	DATA_BLOCK DB381
	TITLE =DBG281M  ELEVATOR 9002 AFTER KILN
	//COPYRIGHT:    (C) 2009  BUHLER AG, CH-9240 UZWIL, SWITZERLAND
	//
	//PRODUCT:      WinCoS_BIW01_09
	//
	//TITLE:        ELEVATOR 9002 AFTER KILN
	//                Machine group DB
	//                Maschinengruppen-DB
	//
	//-------------------------------------------------------------------------
	//
	//IDENT:        AUTHOR:             DEPT:             DATE:
	//
	//P01_DB381.1.0 K.Renz              CSB41             13.Jan.2010
	//              1st Release
	//
	//-------------------------------------------------------------------------
	//
	//PURPOSE:
	//
	//MANUAL :
	//
	//RESTRICTIONS:
	//
	//-------------------------------------------------------------------------
	AUTHOR  : KR
	FAMILY  : USW
	NAME    : DBG281M
	VERSION : 00.00

	FB381
	BEGIN
	      #Gr.Par.ParObjectNo 	:=28100;
	      #Gr.Par.ParIdling      	:=2;
	      #Gr.Par.ParMgr	        :=True;
	      #Gr.Par.ParWgr	        :=False;
	      #Gr.Par.ParGgr	        :=False;
	      #Gr.Par.ParEmptyingTime 	:=0;
	      #Gr.Par.ParHornCode       :=12;
	//Parameter =A-3930-MXZ01MA : ELEVATOR
	      #A_3930_MXZ01MA.Ma.Par.ParObjectNo                                     :=28101;
	      #A_3930_MXZ01MA.Ma.Par.ParWithMon3                                     :=True;
	      #A_3930_MXZ01MA.Ma.Par.ParWithMon4                                     :=True;
	      #A_3930_MXZ01MA.Ma.Par.ParMon1IsHL                                     :=True;
	      #A_3930_MXZ01MA.Ma.Par.ParMon1IsLS                                     :=False;
	      #A_3930_MXZ01MA.Ma.Par.ParMon1StopByFault                              :=True;
	      #A_3930_MXZ01MA.Ma.Par.ParMon2IsLS                                     :=True;
	      #A_3930_MXZ01MA.Ma.Par.ParMon3IsLS                                     :=True;
	      #A_3930_MXZ01MA.Ma.Par.ParMon4AsWarning                                :=False;
	      #A_3930_MXZ01MA.Ma.Par.ParMon4StopByFault                              :=True;
	      #A_3930_MXZ01MA.Ma.Par.ParMon4IsLS                                     :=False;
	      #A_3930_MXZ01MA.Ma.Par.ParWithMon1                                     :=True;
	      #A_3930_MXZ01MA.Ma.Par.ParWithMon5                                     :=False;
	      #A_3930_MXZ01MA.Ma.Par.ParWithMon6                                     :=False;
	      #A_3930_MXZ01MA.Ma.Par.ParEBM                                          :=False;
	      #A_3930_MXZ01MA.Ma.Par.ParMon4IsSM                                     :=True;
	//
	//Parameter A_3930_MXZ01MA.=A-3930-BLH31 : STOWING DETECTOR DISCHARGE
	      #A_3930_MXZ01MA.A_3930_BLH31.Par.ParObjectNo                             :=28102;
	      #A_3930_MXZ01MA.A_3930_BLH31.Par.ParMsgType                              :=7165;
	      #A_3930_MXZ01MA.A_3930_BLH31.Par.ParHornCode                             :=12;
	      #A_3930_MXZ01MA.A_3930_BLH31.Par.ParDelayChange                          :=20;
	      #A_3930_MXZ01MA.A_3930_BLH31.Par.ParDelayCovered                         :=10;
	      #A_3930_MXZ01MA.A_3930_BLH31.Par.ParDelayUncovered                       :=30;
	      #A_3930_MXZ01MA.A_3930_BLH31.Par.ParTimeoutCovered                       :=0;
	      #A_3930_MXZ01MA.A_3930_BLH31.Par.ParTimeoutUncovered                     :=0;
	      #A_3930_MXZ01MA.A_3930_BLH31.Par.ParLogOff                               :=False;
	      #A_3930_MXZ01MA.A_3930_BLH31.Par.Par2WorkingCond                         :=False;
	      #A_3930_MXZ01MA.A_3930_BLH31.Par.ParFaultRetry                           :=False;
	      #A_3930_MXZ01MA.A_3930_BLH31.Par.ParBinLevel                             :=False;
	//
	//Parameter A_3930_MXZ01MA.=A-3930-SHE29 : EMERGENCY-OFF ELEVATOR
	      #A_3930_MXZ01MA.A_3930_SHE29.Par.ParObjectNo                             :=28103;
	      #A_3930_MXZ01MA.A_3930_SHE29.Par.ParMsgType                              :=7136;
	      #A_3930_MXZ01MA.A_3930_SHE29.Par.ParHornCode                             :=12;
	      #A_3930_MXZ01MA.A_3930_SHE29.Par.ParDelayChange                          :=20;
	      #A_3930_MXZ01MA.A_3930_SHE29.Par.ParDelayTrue                            :=10;
	      #A_3930_MXZ01MA.A_3930_SHE29.Par.ParDelayFalse                           :=0;
	      #A_3930_MXZ01MA.A_3930_SHE29.Par.ParTimeoutTrue                          :=0;
	      #A_3930_MXZ01MA.A_3930_SHE29.Par.ParTimeoutFalse                         :=0;
	      #A_3930_MXZ01MA.A_3930_SHE29.Par.ParLogOff                               :=False;
	      #A_3930_MXZ01MA.A_3930_SHE29.Par.Par2WorkingCond                         :=False;
	      #A_3930_MXZ01MA.A_3930_SHE29.Par.ParFaultRetry                           :=False;
	      #A_3930_MXZ01MA.A_3930_SHE29.Par.ParBinLevel                             :=False;
	//
	//Parameter A_3930_MXZ01MA.=A-3930-SHE28 : EMERGENCY-OFF ELEVATOR
	      #A_3930_MXZ01MA.A_3930_SHE28.Par.ParObjectNo                             :=28104;
	      #A_3930_MXZ01MA.A_3930_SHE28.Par.ParMsgType                              :=7136;
	      #A_3930_MXZ01MA.A_3930_SHE28.Par.ParHornCode                             :=12;
	      #A_3930_MXZ01MA.A_3930_SHE28.Par.ParDelayChange                          :=20;
	      #A_3930_MXZ01MA.A_3930_SHE28.Par.ParDelayTrue                            :=10;
	      #A_3930_MXZ01MA.A_3930_SHE28.Par.ParDelayFalse                           :=0;
	      #A_3930_MXZ01MA.A_3930_SHE28.Par.ParTimeoutTrue                          :=0;
	      #A_3930_MXZ01MA.A_3930_SHE28.Par.ParTimeoutFalse                         :=0;
	      #A_3930_MXZ01MA.A_3930_SHE28.Par.ParLogOff                               :=False;
	      #A_3930_MXZ01MA.A_3930_SHE28.Par.Par2WorkingCond                         :=False;
	      #A_3930_MXZ01MA.A_3930_SHE28.Par.ParFaultRetry                           :=False;
	      #A_3930_MXZ01MA.A_3930_SHE28.Par.ParBinLevel                             :=False;
	//
	//Parameter A_3930_MXZ01MA.=A-3930-BSA07 : SPEED CONTROL
	      #A_3930_MXZ01MA.A_3930_BSA07.Par.ParObjectNo                             :=28105;
	      #A_3930_MXZ01MA.A_3930_BSA07.Par.ParMsgType                              :=7135;
	      #A_3930_MXZ01MA.A_3930_BSA07.Par.ParHornCode                             :=12;
	      #A_3930_MXZ01MA.A_3930_BSA07.Par.ParDelayChange                          :=0;
	      #A_3930_MXZ01MA.A_3930_BSA07.Par.ParDelayTrue                            :=10;
	      #A_3930_MXZ01MA.A_3930_BSA07.Par.ParDelayFalse                           :=0;
	      #A_3930_MXZ01MA.A_3930_BSA07.Par.ParTimeoutTrue                          :=50;
	      #A_3930_MXZ01MA.A_3930_BSA07.Par.ParTimeoutFalse                         :=0;
	      #A_3930_MXZ01MA.A_3930_BSA07.Par.ParLogOff                               :=False;
	      #A_3930_MXZ01MA.A_3930_BSA07.Par.Par2WorkingCond                         :=True;
	      #A_3930_MXZ01MA.A_3930_BSA07.Par.ParFaultRetry                           :=False;
	      #A_3930_MXZ01MA.A_3930_BSA07.Par.ParBinLevel                             :=False;
	//
	//Parameter A_3930_MXZ01MA.=A-3930-MXZ01 : ELEVATOR
	      #A_3930_MXZ01MA.A_3930_MXZ01.Par.ParObjectNo                             :=28106;
	      #A_3930_MXZ01MA.A_3930_MXZ01.Par.ParMsgType                              :=7053;
	      #A_3930_MXZ01MA.A_3930_MXZ01.Par.ParHornCode                             :=12;
	      #A_3930_MXZ01MA.A_3930_MXZ01.Par.ParMonTime                              :=20;
	      #A_3930_MXZ01MA.A_3930_MXZ01.Par.ParStartingTime                         :=20;
	      #A_3930_MXZ01MA.A_3930_MXZ01.Par.ParStoppingTime                         :=0;
	      #A_3930_MXZ01MA.A_3930_MXZ01.Par.ParIdlingTime                           :=0;
	      #A_3930_MXZ01MA.A_3930_MXZ01.Par.ParDelayTime                            :=10;
	      #A_3930_MXZ01MA.A_3930_MXZ01.Par.ParLogOff                               :=False;
	      #A_3930_MXZ01MA.A_3930_MXZ01.Par.ParManual                               :=True;
	      #A_3930_MXZ01MA.A_3930_MXZ01.Par.ParRestartDelay                         :=False;
	      #A_3930_MXZ01MA.A_3930_MXZ01.Par.Par2Speed                               :=False;
	      #A_3930_MXZ01MA.A_3930_MXZ01.Par.ParHeavyStartup                         :=False;
	//
	//
	//Parameter =A-3932-MXZ01MA : FILTER ASPIRATION ELEVATOR
	      #A_3932_MXZ01MA.Ma.Par.ParObjectNo                                     :=28107;
	      #A_3932_MXZ01MA.Ma.Par.ParWithAirlock                                  :=False;
	      #A_3932_MXZ01MA.Ma.Par.ParWithFan                                      :=True;
	      #A_3932_MXZ01MA.Ma.Par.ParWithFilter                                   :=True;
	      #A_3932_MXZ01MA.Ma.Par.ParWithARF                                      :=False;
	      #A_3932_MXZ01MA.Ma.Par.ParWithLSDoor                                   :=False;
	      #A_3932_MXZ01MA.Ma.Par.ParWithPressure                                 :=False;
	      #A_3932_MXZ01MA.Ma.Par.ParWithHLAirlock                                :=False;
	      #A_3932_MXZ01MA.Ma.Par.ParWithDischarger                               :=False;
	      #A_3932_MXZ01MA.Ma.Par.ParVibroOnTime                                  :=0;
	      #A_3932_MXZ01MA.Ma.Par.ParVibroOffTime                                 :=0;
	//
	//Parameter A_3932_MXZ01MA.=A-3932-MXZ01 : FAN DRIVE
	      #A_3932_MXZ01MA.A_3932_MXZ01.Par.ParObjectNo                             :=28108;
	      #A_3932_MXZ01MA.A_3932_MXZ01.Par.ParMsgType                              :=7053;
	      #A_3932_MXZ01MA.A_3932_MXZ01.Par.ParHornCode                             :=12;
	      #A_3932_MXZ01MA.A_3932_MXZ01.Par.ParMonTime                              :=20;
	      #A_3932_MXZ01MA.A_3932_MXZ01.Par.ParStartingTime                         :=20;
	      #A_3932_MXZ01MA.A_3932_MXZ01.Par.ParStoppingTime                         :=0;
	      #A_3932_MXZ01MA.A_3932_MXZ01.Par.ParIdlingTime                           :=0;
	      #A_3932_MXZ01MA.A_3932_MXZ01.Par.ParDelayTime                            :=10;
	      #A_3932_MXZ01MA.A_3932_MXZ01.Par.ParLogOff                               :=False;
	      #A_3932_MXZ01MA.A_3932_MXZ01.Par.ParManual                               :=True;
	      #A_3932_MXZ01MA.A_3932_MXZ01.Par.ParRestartDelay                         :=False;
	      #A_3932_MXZ01MA.A_3932_MXZ01.Par.Par2Speed                               :=False;
	      #A_3932_MXZ01MA.A_3932_MXZ01.Par.ParHeavyStartup                         :=False;
	//
	//Parameter A_3932_MXZ01MA.=A-3931-KFC10 : FILTER ASPIRATION
	      #A_3932_MXZ01MA.A_3931_KFC10.Par.ParObjectNo                             :=28109;
	      #A_3932_MXZ01MA.A_3931_KFC10.Par.ParMsgType                              :=7002;
	      #A_3932_MXZ01MA.A_3931_KFC10.Par.ParHornCode                             :=12;
	      #A_3932_MXZ01MA.A_3931_KFC10.Par.ParOnTime                               :=50;
	      #A_3932_MXZ01MA.A_3931_KFC10.Par.ParOffTime                              :=0;
	      #A_3932_MXZ01MA.A_3931_KFC10.Par.ParIdlingTime                           :=3000;
	      #A_3932_MXZ01MA.A_3931_KFC10.Par.ParDelayTime                            :=0;
	      #A_3932_MXZ01MA.A_3931_KFC10.Par.ParLogOff                               :=False;
	      #A_3932_MXZ01MA.A_3931_KFC10.Par.ParManual                               :=True;
	      #A_3932_MXZ01MA.A_3931_KFC10.Par.ParContinuous                           :=True;
	      #A_3932_MXZ01MA.A_3931_KFC10.Par.ParPulse                                :=False;
	      #A_3932_MXZ01MA.A_3931_KFC10.Par.ParPulsing                              :=False;
	      #A_3932_MXZ01MA.A_3931_KFC10.Par.ParFilter                               :=True;
	//
	//
	//Parameter =A-3930-KCL01 : RESET DISTURBANCE ELEVATOR
	      #A_3930_KCL01.Par.ParObjectNo                             :=28110;
	      #A_3930_KCL01.Par.ParMsgType                              :=7154;
	      #A_3930_KCL01.Par.ParHornCode                             :=12;
	      #A_3930_KCL01.Par.ParDelayChange                          :=20;
	      #A_3930_KCL01.Par.ParDelayTrue                            :=10;
	      #A_3930_KCL01.Par.ParDelayFalse                           :=0;
	      #A_3930_KCL01.Par.ParTimeoutTrue                          :=0;
	      #A_3930_KCL01.Par.ParTimeoutFalse                         :=0;
	      #A_3930_KCL01.Par.ParLogOff                               :=False;
	      #A_3930_KCL01.Par.Par2WorkingCond                         :=False;
	      #A_3930_KCL01.Par.ParFaultRetry                           :=False;
	      #A_3930_KCL01.Par.ParBinLevel                             :=False;
	//
	//
	//Parameter =A-3930-PII24 : CURRENT MEASURING
	      #A_3930_PII24.Par.ParObjectNo                             :=28111;
	      #A_3930_PII24.Par.ParHornCode                             :=12;
	      #A_3930_PII24.Par.ParMsgType                              :=7252;
	      #A_3930_PII24.Par.ParUnitsByZeroDigit                     :=L#0;
	      #A_3930_PII24.Par.ParUnitsByMaxDigit                      :=L#27648;
	      #A_3930_PII24.Par.ParUnitsBy100Pc                         :=L#10000;
	      #A_3930_PII24.Par.ParDelayTimeDown                        :=10;
	      #A_3930_PII24.Par.ParDelayTimeUp                          :=10;
	      #A_3930_PII24.Par.ParDelayTime                            :=0;
	      #A_3930_PII24.Par.ParLimitLL                              :=L#0;
	      #A_3930_PII24.Par.ParLimitL                               :=L#2000;
	      #A_3930_PII24.Par.ParLimitH                               :=L#10000;
	      #A_3930_PII24.Par.ParLimitHH                              :=L#10100;
	      #A_3930_PII24.Par.ParMonTimeLL                            :=0;
	      #A_3930_PII24.Par.ParMonTimeL                             :=50;
	      #A_3930_PII24.Par.ParMonTimeMid                           :=0;
	      #A_3930_PII24.Par.ParMonTimeH                             :=30;
	      #A_3930_PII24.Par.ParMonTimeHH                            :=0;
	      #A_3930_PII24.Par.ParLogOff                               :=False;
	      #A_3930_PII24.Par.ParValueByUser                          :=False;
	      #A_3930_PII24.Par.ParLimitsPc                             :=True;
	      #A_3930_PII24.Par.ParWago                                 :=False;
	      #A_3930_PII24.Par.ParNoHornByWarning                      :=True;
	      #A_3930_PII24.Par.ParWarningLL                            :=False;
	      #A_3930_PII24.Par.ParWarningL                             :=False;
	      #A_3930_PII24.Par.ParWarningMid                           :=False;
	      #A_3930_PII24.Par.ParWarningH                             :=False;
	      #A_3930_PII24.Par.ParWarningHH                            :=False;
	      #A_3930_PII24.Par.ParPreAlarmLL                           :=False;
	      #A_3930_PII24.Par.ParPreAlarmL                            :=False;
	      #A_3930_PII24.Par.ParPreAlarmMid                          :=False;
	      #A_3930_PII24.Par.ParPreAlarmH                            :=False;
	      #A_3930_PII24.Par.ParPreAlarmHH                           :=False;
	//
	//
	//Parameter =A-3930-QYS30 : EXPLOSION VENT ELEVATOR
	      #A_3930_QYS30.Par.ParObjectNo                             :=28112;
	      #A_3930_QYS30.Par.ParMsgType                              :=7136;
	      #A_3930_QYS30.Par.ParHornCode                             :=12;
	      #A_3930_QYS30.Par.ParDelayChange                          :=20;
	      #A_3930_QYS30.Par.ParDelayTrue                            :=10;
	      #A_3930_QYS30.Par.ParDelayFalse                           :=0;
	      #A_3930_QYS30.Par.ParTimeoutTrue                          :=0;
	      #A_3930_QYS30.Par.ParTimeoutFalse                         :=0;
	      #A_3930_QYS30.Par.ParLogOff                               :=False;
	      #A_3930_QYS30.Par.Par2WorkingCond                         :=False;
	      #A_3930_QYS30.Par.ParFaultRetry                           :=False;
	      #A_3930_QYS30.Par.ParBinLevel                             :=False;
	//
	//
	//Parameter =A-3930-BZ08CU : NO FAILURE ELEVATOR
	      #A_3930_BZ08CU.Par.ParObjectNo                             :=28113;
	      #A_3930_BZ08CU.Par.ParMsgType                              :=7154;
	      #A_3930_BZ08CU.Par.ParHornCode                             :=12;
	      #A_3930_BZ08CU.Par.ParDelayChange                          :=20;
	      #A_3930_BZ08CU.Par.ParDelayTrue                            :=10;
	      #A_3930_BZ08CU.Par.ParDelayFalse                           :=0;
	      #A_3930_BZ08CU.Par.ParTimeoutTrue                          :=0;
	      #A_3930_BZ08CU.Par.ParTimeoutFalse                         :=0;
	      #A_3930_BZ08CU.Par.ParLogOff                               :=False;
	      #A_3930_BZ08CU.Par.Par2WorkingCond                         :=False;
	      #A_3930_BZ08CU.Par.ParFaultRetry                           :=False;
	      #A_3930_BZ08CU.Par.ParBinLevel                             :=False;
	//
	//
	END_DATA_BLOCK
